(* IEC 61131-3 sources: RL_MAR/experiments/comparison/llm4plc/results/deepseek-ai-DeepSeek-V3.2_20260506_104945/20260506_112754, 1 file *)

(* ---- generated_code_iteration_0.st ---- *)
START_ST
FUNCTION_BLOCK CottonCandyMachine
VAR_INPUT
    SugarLevel : REAL;
    SpinningSpeed : INT;
END_VAR
VAR_OUTPUT
    SugarFeeder : BOOL;
    MotorSpeed : INT;
END_VAR

(* State 0: OPERATE - Continuous evaluation of inputs to set outputs *)
SugarFeeder := (SugarLevel < 10.0);
IF SpinningSpeed > 0 THEN
    MotorSpeed := SpinningSpeed;
ELSE
    MotorSpeed := 0;
END_IF;

END_FUNCTION_BLOCK
END_ST
